// TIA Portal V17 export
// export: Created 2024-08-07T21:44:11.5414672Z, ExportSetting WithDefaults, DisplayName Totally Integrated Automation Portal, DisplayVersion V17 Update 7, DisplayName TIA Portal Openness, DisplayVersion V17 Update 7, DisplayName TIA Portal Version Control Interface, DisplayVersion V17, DisplayName SINAMICS Startdrive Advanced, DisplayVersion V17 SP2, DisplayName SINAMICS Startdrive G110M, G120, G120C, G120D, G120P, G115D, DisplayVersion V17 SP2, DisplayName SINAMICS Startdrive G130, G150, S120, S150, SINAMICS MV, S210, DisplayVersion V17 SP2, DisplayName STEP 7 Professional, DisplayVersion V17 Update 7, DisplayName STEP 7 Safety, DisplayVersion V17 Update 6, DisplayName WinCC Advanced / Unified PC, DisplayVersion V17 Update 7
DATA_BLOCK "5. Call_M005_VARIABILITY_DB"   // DB2005
VERSION : 0.1
// stored: AutoNumber false, DBAccessibleFromOPCUA true, DBAccessibleFromWebserver true, InstanceOfName 5. Call_M005_VARIABILITY, InstanceOfType FB
"5. Call_M005_VARIABILITY"
   // VAR_INPUT
   //    equipmentVariability : WString;
   //    errorDInt : Array[1..32] of DInt;
   //    errorWString : Array[1..32] of WString;
   //    x : Bool;
   // END_VAR
   // VAR
   //    variabilityIndex { ExternalAccessible := 'False'; ExternalVisible := 'False'; ExternalWritable := 'False'} : Array[1..32] of WString[1];
   //    actualValue : Array[1..32] of DInt;
   //    timestamp : DTL;
   //    timestampStr : Struct
   //       year : WString;
   //       month : WString;
   //       day : WString;
   //       hour : WString;
   //       minute : WString;
   //       second : WString;
   //    END_STRUCT;
   //    datestring : String;
   // END_VAR
BEGIN
END_DATA_BLOCK
